// TwinCAT 3 PLC project PID_Projekt
// ProgramVersion: 3.1.4023.0
// libraries:
//   Tc2_ControllerToolbox, * (Beckhoff Automation GmbH)
//   Tc2_MC2, * (Beckhoff Automation GmbH)
//   Tc2_Standard, * (Beckhoff Automation GmbH)
//   Tc2_System, * (Beckhoff Automation GmbH)
//   Tc3_Module, * (Beckhoff Automation GmbH)
// project tree:
//   DUTs/ state.TcDUT
//   / GlobalTextList.TcGTLO, PlcTask.TcTTO, Visualisierungsmanager.TcVMO (not stored)
//   GVLs/ GVL.TcGVL
//   POUs/ MAIN.TcPOU, Signalersteller.TcPOU
// real-time tasks:
//   TASK PlcTask: cycle T#5ms, priority 20, ADS port 350
// motion (NC):
//   TASK NC-Task 1 SAF: cycle T#2ms, priority 4, ADS port 501
//   TASK NC-Task 1 SVB: cycle T#10ms, priority 8, ADS port 511
//   AXIS Achse 1 (id 1) // MyAxis
//     OtherSettings: AllowMotionCmdToSlave=true
//     encoder EncType=1
//     drive DrvType=5
//       Analog: TorqueSetpointScale=10, ScaleFactorActTorque=0.1
//       TimeComp: TaskDelayCycles=1
//     controller CtrType=1
//       CtrPara: PriorControlFactor=1
//         Observer: BandWidth=20
// variable links:
//   PID_Projekt/PID_Projekt Instance <-> NC-Task 1 SAF/Axes/Achse 1
//     PlcTask Inputs/MAIN.axis.NcToPlc <-> Outputs/ToPlc
//     PlcTask Outputs/MAIN.axis.PlcToNc <-> Inputs/FromPlc

CONFIGURATION PID_Projekt
    RESOURCE PLC ON TwinCAT3
        TASK PlcTask(INTERVAL := T#5ms, PRIORITY := 20);
        PROGRAM MAIN WITH PlcTask : MAIN;
    END_RESOURCE
END_CONFIGURATION

// ---- DUTs/state.TcDUT
TYPE state :
(
	INIT,
	POWER_ON,
	MOVE_ON,
	ERROR,
	P_RESET
)UDINT;
END_TYPE

// ---- GVLs/GVL.TcGVL
{attribute 'qualified_only'}
VAR_GLOBAL
	
	MC_MoveAbsolute: MC_MoveAbsolute;
	MC_MoveAbsolute_output: ST_McOutputs;
END_VAR

// ---- POUs/MAIN.TcPOU
PROGRAM MAIN
VAR
    axis: AXIS_REF;
	MC_ReadActualPosition: MC_ReadActualPosition;
	MC_ReadActualVelocity: MC_ReadActualVelocity;
	state: state;
	
	reset_output:ST_McOutputs;
	axis_Reset: MC_Reset;
	ReadP_Valid:BOOL;
	ReadV_Valid:BOOL;
	Position: LREAL;
	Velocity: LREAL;
	power1: MC_Power;
	power1_output:ST_McOutputs;
END_VAR

// Programmablauf mittels Zustandsautomat
CASE state OF
	
	INIT:
		GVL.MC_MoveAbsolute.Execute := FALSE;
		Power1.Enable:=FALSE;
		axis_Reset.Execute:=FALSE;
		state := POWER_ON;
	
	POWER_ON:
		Power1.Enable := TRUE;
		IF power1_output.Done = TRUE THEN
			state := MOVE_ON;
		ELSIF power1_output.Done = FALSE THEN
			state := POWER_ON;
		END_IF
		IF axis.Status.Error THEN
			state := ERROR;
		END_IF
 
	MOVE_ON:
		IF GVL.MC_MoveAbsolute_output.Busy = FALSE THEN	
			GVL.MC_MoveAbsolute.Velocity := 10;
			GVL.MC_MoveAbsolute.Execute := TRUE;
			//state := MOVE_ON;
		END_IF
		
		IF GVL.MC_MoveAbsolute.Done THEN
			state := INIT;
		END_IF
		
		IF axis.Status.Error THEN
			state := ERROR;
		END_IF
		
	ERROR:
		GVL.MC_MoveAbsolute.Execute:=FALSE;
		IF NOT axis.Status.Coupled THEN
			IF axis.Status.Error THEN
				state := P_RESET;	
			ELSE
				state := INIT;
			END_IF
		END_IF
		
	P_RESET:
		axis_Reset.Execute := TRUE;
		GVL.MC_MoveAbsolute.Execute:=FALSE;
			
			IF axis_Reset.Done  THEN
				state := INIT;
			ELSIF axis_Reset.Error  THEN
				state := INIT; 
			END_IF
END_CASE

axis();
Signalersteller();
power();
MoveAbsolute();
ReadP_V();
reset();

ACTION MoveAbsolute:
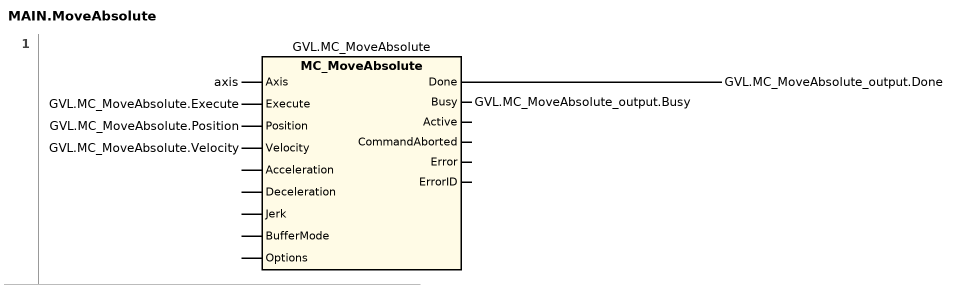
// NETWORK 1
GVL.MC_MoveAbsolute(
    Axis := axis,
    Execute := GVL.MC_MoveAbsolute.Execute,
    Position := GVL.MC_MoveAbsolute.Position,
    Velocity := GVL.MC_MoveAbsolute.Velocity,
    Busy => GVL.MC_MoveAbsolute_output.Busy); // MC_MoveAbsolute
GVL.MC_MoveAbsolute_output.Done := GVL.MC_MoveAbsolute.Done;
END_ACTION

ACTION PID:
// NETWORK 1
END_ACTION

ACTION Power:
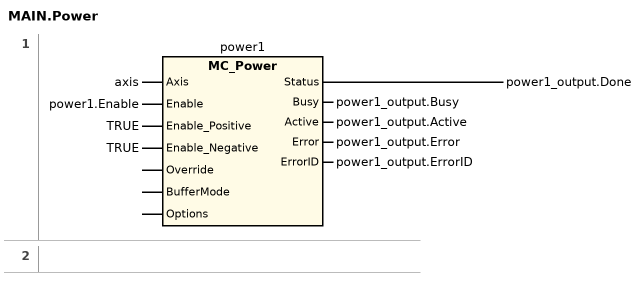
// NETWORK 1
power1(
    Axis := axis,
    Enable := power1.Enable,
    Enable_Positive := TRUE,
    Enable_Negative := TRUE,
    Busy => power1_output.Busy,
    Active => power1_output.Active,
    Error => power1_output.Error,
    ErrorID => power1_output.ErrorID); // MC_Power
power1_output.Done := power1.Status;

// NETWORK 2
END_ACTION

ACTION ReadP_V:
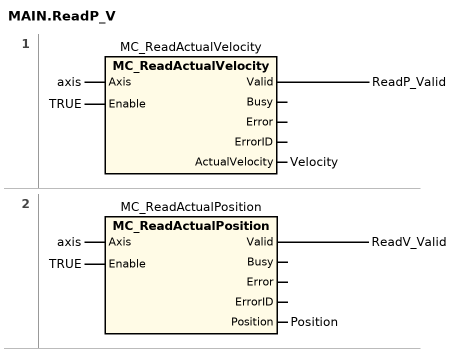
// NETWORK 1
MC_ReadActualVelocity(Axis := axis, Enable := TRUE, ActualVelocity => Velocity);
ReadP_Valid := MC_ReadActualVelocity.Valid;

// NETWORK 2
MC_ReadActualPosition(Axis := axis, Enable := TRUE, Position => Position);
ReadV_Valid := MC_ReadActualPosition.Valid;
END_ACTION

ACTION Reset:
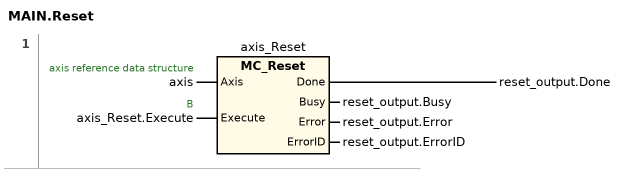
// NETWORK 1
//   axis: axis reference data structure
//   axis_Reset.Execute: B
axis_Reset(
    Axis := axis,
    Execute := axis_Reset.Execute,
    Busy => reset_output.Busy,
    Error => reset_output.Error,
    ErrorID => reset_output.ErrorID); // MC_Reset
reset_output.Done := axis_Reset.Done;
END_ACTION

END_PROGRAM

// ---- POUs/Signalersteller.TcPOU
PROGRAM Signalersteller

VAR
	TP_Timer: TP;
	TON_Timer: TON;
	PWM_On: BOOL := 0;
	TP_Timer_Output: BOOL := 0;
	TON_Timer_Output: BOOL := 0;
	TON_Time: TIME;
	TP_Time: TIME;
	Timer_Start: BOOL := 1;
	SignalToggle: BOOL := FALSE;
	SignalPWM: INT;
	MODE: INT := 1;
END_VAR

IF TON_Time>=T#4S THEN
	Timer_Start:=FALSE;
END_IF
TON_Timer(IN:= Timer_Start, PT:= T#4S, Q=> PWM_On, ET=> TON_Time);
IF Timer_Start=FALSE THEN
	Timer_Start:=TRUE;
END_IF

TP_Timer(IN:= PWM_On, PT:= T#2S, Q=> TP_Timer_Output, ET=> TP_Time);

IF TP_Timer_Output THEN
	GVL.MC_MoveAbsolute.Position := 5;
ELSE GVL.MC_MoveAbsolute.Position := 0;
END_IF

//IF MODE=0 THEN
//	MC_MoveAbsolute.Position := Signal;
//ELSIF MODE = 1 THEN
//	MC_MoveAbsolute.Position := SignalPWM;
//END_IF

//IF Signal >= 10 THEN
//	SignalToggle := TRUE;
//	SignalPWM := 10;
//ELSIF Signal <= 0 THEN
//	SignalToggle := FALSE;
//	SignalPWM:=0;
//END_IF

//IF SignalToggle = FALSE THEN 
//	Signal := Signal + 0.01;
//ELSIF SignalToggle = TRUE THEN
//	Signal := Signal - 0.01;
//END_IF

END_PROGRAM

// ---- GlobalTextList.TcGTLO
TEXTLIST GlobalTextList
  95 = 'PowerEnable'
END_TEXTLIST
